FUNCTION_BLOCK T_ClassThatRaisesNotifications
VAR_INPUT
END_VAR
VAR_OUTPUT
END_VAR
VAR
    OnPbPressed_Notification : T_Notification := (NotificationId := E_Test_NotificationId.OnPbPressed_Notification); // This name used to identify the notification
    PbIdentifier : STRING := 'CP23';
END_VAR

PROPERTY OnPressedNotification : I_Notification
GET
OnPressedNotification := OnPbPressed_Notification;
END_GET
END_PROPERTY

METHOD RaiseOnPbPressedNotification
VAR_INPUT
END_VAR
OnPbPressed_Notification.Args
    .Clear()
    .Add_STRING(PbIdentifier);
OnPbPressed_Notification.Raise();
END_METHOD

END_FUNCTION_BLOCK

(* stored: Version 1.1.0.1, ProductVersion 3.1.4024.5
   POU T_ClassThatRaisesNotifications: Id {c11d4f62-058c-42a7-933f-c523f0c1c82d}, SpecialFunc None
   Property OnPressedNotification: Id {0a0297c3-1d14-421b-907e-fde2e3a09660}
   Get Get: Id {7eecedc7-374a-4e06-8352-9faeb9bd5856}
   Method RaiseOnPbPressedNotification: Id {804c7876-622a-42b7-ad87-f6ef097ca46f} *)
